(* PLC project OpenPLC_Testing, Binary-6 PiPLC_DemoProduct 1, author Chrismettal *)
(* stored: creationDateTime 2023-12-08T21:28:31, companyURL Binary-6.de, modificationDateTime 2023-12-12T16:54:12, language en-US *)

PROGRAM MAIN
  VAR
    Input_I1 AT %IX0.0 : BOOL;
    Input_I2 AT %IX0.1 : BOOL;
    Input_I3 AT %IX0.2 : BOOL;
    Input_I4 AT %IX0.3 : BOOL;
    Input_I5 AT %IX0.4 : BOOL;
    Input_I6 AT %IX0.5 : BOOL;
    Input_I7 AT %IX0.6 : BOOL;
    Input_I8 AT %IX0.7 : BOOL;
    Output_Q1 AT %QX0.0 : BOOL;
    Output_Q2 AT %QX0.1 : BOOL;
    Output_Q3 AT %QX0.2 : BOOL;
    Output_Q4 AT %QX0.3 : BOOL;
    Output_Q5 AT %QX0.4 : BOOL;
    Output_Q6 AT %QX0.5 : BOOL;
    Output_Q7 AT %QX0.6 : BOOL;
    Output_Q8 AT %QX0.7 : BOOL;
    PWM_0 AT %QW0 : WORD;
    PWM_1 AT %QW1 : WORD;
  END_VAR
  VAR
    InitDone : BOOL := FALSE;
  END_VAR
  VAR
    ModIO_Q1 AT %QX100.0 : BOOL;
    ModIO_Q2 AT %QX100.1 : BOOL;
    ModIO_Q3 AT %QX100.2 : BOOL;
    ModIO_Q4 AT %QX100.3 : BOOL;
  END_VAR

            (* This is a testing program to test most functions on a PiPLC                                      *)
(* Make sure to activate the "Binary-6 PiPLC" hardware layer on your PLC before uploading this code *)

IF NOT InitDone THEN
  (* Oneshots at init *)

  (* PWM demo, set an arbitrary duty cycle to PWM outputs. *)
  PWM_0 := 32760; (* ~50% Duty Cycle *)
  PWM_1 := 8000; (* ~12% Duty Cycle *)
    
  (* Set InitDone so we execute cyclic tasks starting next scan *)
  InitDone := TRUE;

ELSE
  (* Cyclic calls after init oneshots*)
  
  (* Digital I/O demo. Pass Ix to Qx live *)
  Output_Q1 := Input_I1;
  Output_Q2 := Input_I2;
  Output_Q3 := Input_I3;
  Output_Q4 := Input_I4;
  Output_Q5 := Input_I5;
  Output_Q6 := Input_I6;
  Output_Q7 := Input_I7;
  Output_Q8 := Input_I8;

  (* Write out Modbus outputs *)
  ModIO_Q1  := Input_I1;
  ModIO_Q2  := Input_I2;
  ModIO_Q3  := Input_I3;
  ModIO_Q4  := Input_I4;

  (* TODO 1-Wire demo here *)
  
  (* TODO I2C demo here *)
  
END_IF;

          
END_PROGRAM

CONFIGURATION Config0
  RESOURCE Res0 ON PLC
    TASK PlcTask(INTERVAL := T#20ms, PRIORITY := 0);
    PROGRAM instance0 WITH PlcTask : MAIN;
  END_RESOURCE
END_CONFIGURATION
